FUNCTION F_Get_Parent_Path : T_MAXSTRING
VAR_INPUT
	child_path: T_MAXSTRING;
END_VAR
VAR
	_output_string: T_MAXSTRING;
	_dot_position: INT;
END_VAR

WHILE TRUE DO
	_dot_position := FIND(child_path, '.');	
	
	IF _dot_position = 0 THEN
		_output_string := DELETE(_output_string, 1, LEN(_output_string));
		F_Get_Parent_Path := _output_string;
		RETURN;
	END_IF
	
	_output_string := CONCAT(_output_string, LEFT(child_path, _dot_position));
		
	child_path := DELETE(child_path, _dot_position, 1);
	

END_WHILE

END_FUNCTION

(* stored: Version 1.1.0.1, ProductVersion 3.1.4024.12
   POU F_Get_Parent_Path: Id {58bf5ad2-8079-4d52-aa81-2c75d9f51c07}, SpecialFunc None *)
